Yaskawa INFORM job: X2_7,2(150,-90).JBI

/JOB
//NAME X2_7,2(150,-90)
//POS
///NPOS 31,31,31,3,0,0
///TOOL 0
///POSTYPE PULSE
///PULSE
C00000=1903,-101039,-123464,18,98414,-30
C00001=-37629,-83041,-126142,-12125,101236,40991
C00002=-120710,-114236,-128002,161,94425,119
C00003=-120626,-97263,-85517,147,77002,126
C00004=-120624,-90603,-79512,147,76729,126
C00005=-120619,-87609,-75876,147,76029,126
C00006=-120612,-86998,-74157,145,75286,128
C00007=-120630,-84931,-74575,148,76604,124
C00008=-120635,-82574,-72610,148,76606,123
C00009=-120636,-81941,-72345,149,76768,122
C00010=-120635,-82574,-72610,148,76606,123
C00011=-120623,-96358,-82912,147,75863,125
C00012=-120643,-96591,-84648,150,76812,120
C00013=-120640,-89962,-78640,150,76521,120
C00014=-120640,-87399,-76229,150,76354,120
C00015=-120632,-86713,-74265,149,75498,122
C00016=-120630,-86551,-75442,148,76306,123
C00017=-120611,-84912,-73908,144,76204,130
C00018=-120616,-83150,-73182,145,76663,128
C00019=-120611,-84912,-73908,144,76204,130
C00020=-120607,-95796,-83038,144,76230,131
C00021=-120623,-87424,-78135,4974,77554,-1131
C00022=-120623,-86585,-74968,5002,76042,-1192
C00023=-120623,-87260,-75250,5004,75869,-1199
C00024=-120623,-87371,-75295,5004,75876,-1199
C00025=-120621,-87568,-75289,5005,75773,-1205
C00026=-120621,-87481,-75230,5007,75741,-1203
C00027=-120623,-86357,-74872,5001,76100,-1190
C00028=-120623,-87221,-78171,4972,77680,-1126
C00029=-120710,-114236,-128002,161,94425,119
C00030=1903,-101039,-123464,18,98414,-30
BC00000=178026,670300,1070054
BC00001=191697,740247,974662
BC00002=183510,780543,1070054
BC00003=183510,787889,1070054
BC00004=183510,787889,1070054
BC00005=183510,787889,1070054
BC00006=183510,787889,1070054
BC00007=183510,787889,1070054
BC00008=183510,787889,1070054
BC00009=183510,787889,1070054
BC00010=183510,787889,1070054
BC00011=183510,787889,1070054
BC00012=246548,789373,1069572
BC00013=246548,789373,1069572
BC00014=246548,789373,1069572
BC00015=246548,789373,1069572
BC00016=246548,789373,1069572
BC00017=246548,789373,1069572
BC00018=246548,789373,1069572
BC00019=246548,789373,1069572
BC00020=246548,789373,1069572
BC00021=173122,786192,1075175
BC00022=173821,790731,1071691
BC00023=174101,792546,1063067
BC00024=178879,792629,1063203
BC00025=232874,792823,1063865
BC00026=237653,792774,1063847
BC00027=237373,790958,1072470
BC00028=236673,786420,1075175
BC00029=183510,780543,1070054
BC00030=178026,670300,1070054
EC00000=1330261,-556475
EC00001=1330261,-556473
EC00002=1330261,-556475
EC00003=1330261,-556475
EC00004=1330261,-556475
EC00005=1330261,-556475
EC00006=1330261,-556475
EC00007=1330261,-556475
EC00008=1330261,-556475
EC00009=1330261,-556475
EC00010=1330261,-556475
EC00011=1330261,-556475
EC00012=1330261,-556475
EC00013=1330261,-556475
EC00014=1330261,-556475
EC00015=1330261,-556475
EC00016=1330261,-556475
EC00017=1330261,-556475
EC00018=1330261,-556475
EC00019=1330261,-556475
EC00020=1330261,-556475
EC00021=1330261,-556475
EC00022=1330261,-556475
EC00023=1330261,-556475
EC00024=1330261,-556475
EC00025=1330261,-556475
EC00026=1330261,-556475
EC00027=1330261,-556475
EC00028=1330261,-556475
EC00029=1330261,-556475
EC00030=1330261,-556475
///POSTYPE BASE
///RECTAN
///RCONF 0,0,0,0,0,0,0,0,0,0,0,0,0,0,0,0,0,0,0,0,0,0,0,0
P00006=0.222,-3.123,-1.508,0.0000,0.0000,0.0000
P00021=-0.225,-6.128,-0.405,0.0000,0.0000,0.0000
P00022=0.222,-3.123,-1.508,0.0000,0.0000,0.0000
//INST
///DATE 2024/04/06 15:25
///ATTR SC,RW
///GROUP1 RB1,BS1
///GROUP2 ST1
NOP
'X2_7,2(150,-90)
MOVJ C00000 BC00000 VJ=100.00  +MOVJ EC00000 VJ=100.00
CALL JOB:CLEAN-R1_KM_NEW
MOVJ C00001 BC00001 VJ=100.00  +MOVJ EC00001 VJ=100.00
MOVJ C00002 BC00002 VJ=100.00  +MOVJ EC00002 VJ=100.00
'Path S3593
SFTOF3D
MOVJ C00003 BC00003 VJ=100.00  +MOVJ EC00003 VJ=100.00
MOVL C00004 BC00004 V=666.7  +MOVJ EC00004 VJ=100.00
SMOVL C00005 BC00005 V=166.7  +MOVJ EC00005
SREFP 3 C00006 BC00006  +REFP EC00006
CALL JOB:SEARCH-R1-S13D
SET P021 P006
SFTON3D P021
SMOVL C00007 BC00007 V=250.0  +MOVJ EC00007
SMOVL C00008 BC00008 V=166.7  +MOVJ EC00008
SREFP 3 C00009 BC00009  +REFP EC00009
CALL JOB:SEARCH-R1-S13D
SET P021 P006
SFTON3D P021
SMOVL C00010 BC00010 V=250.0  +MOVJ EC00010
MOVL C00011 BC00011 V=1000.0  +MOVJ EC00011 VJ=100.00
'EndPath S3593
'Path S4333
SFTOF3D
MOVJ C00012 BC00012 VJ=100.00  +MOVJ EC00012 VJ=100.00
MOVL C00013 BC00013 V=666.7  +MOVJ EC00013 VJ=100.00
SMOVL C00014 BC00014 V=166.7  +MOVJ EC00014
SREFP 3 C00015 BC00015  +REFP EC00015
CALL JOB:SEARCH-R1-S13D
SET P022 P006
SFTON3D P022
SMOVL C00016 BC00016 V=250.0  +MOVJ EC00016
SMOVL C00017 BC00017 V=166.7  +MOVJ EC00017
SREFP 3 C00018 BC00018  +REFP EC00018
CALL JOB:SEARCH-R1-S13D
SET P022 P006
SFTON3D P022
SMOVL C00019 BC00019 V=250.0  +MOVJ EC00019
MOVL C00020 BC00020 V=1000.0  +MOVJ EC00020 VJ=100.00
'EndPath S4333
'Path W3596
SFTOF3D
SFTON3D P021
MOVJ C00021 BC00021 VJ=100.00  +MOVJ EC00021 VJ=100.00
SMOVL C00022 BC00022 V=666.7  +MOVJ EC00022
SMOVL C00023 BC00023 V=166.7 PL=0  +MOVJ EC00023
MACRO1 MJ#(0) ARGF21
ARCON
SMOVL C00024 BC00024 V=9.2  +MOVJ EC00024
SMOVL C00025 BC00025 V=9.2  +MOVJ EC00025
SMOVL C00026 BC00026 V=9.2  +MOVJ EC00026
ARCOF
SMOVL C00027 BC00027 V=800.0  +MOVJ EC00027
SMOVL C00028 BC00028 V=1000.0  +MOVJ EC00028
SFTOF3D
'EndPath W3596
MOVJ C00029 BC00029 VJ=100.00  +MOVJ EC00029 VJ=100.00
MOVJ C00030 BC00030 VJ=100.00  +MOVJ EC00030 VJ=100.00
END
